FUNCTION_BLOCK FB_ProcessSimulation
VAR_INPUT
	bEnable: BOOL;
	
	bRotateTable: BOOL;
	bLinearSliderMoveToPick : BOOL;
	bLinearSliderMoveToPlace : BOOL;
	
	tPartSensorDelay: TIME;
	tLinearSliderPickPosSensorDelay : TIME;
	tLinearSliderPlacePosSensorDelay : TIME;
END_VAR
VAR_OUTPUT
	bPartSensorSignal: BOOL;
	bLinearSliderPickPosSensorSignal: BOOL;
	bLinearSliderPlacePosSensorSignal: BOOL; 
END_VAR
VAR
	fbPartSensorDelayTmr: TON;
	fbLinearSliderPickPosSensorDelayTmr: TON;
	fbLinearSliderPlacePosSensorDelayTmr: TON;
END_VAR

fbPartSensorDelayTmr(IN:= bEnable AND bRotateTable, 
					PT:= tPartSensorDelay, 
					Q=> bPartSensorSignal, ET=> );
					
fbLinearSliderPickPosSensorDelayTmr(IN:= bEnable AND bLinearSliderMoveToPick, 
									PT:= tLinearSliderPickPosSensorDelay, 
									Q=> bLinearSliderPickPosSensorSignal, ET=> );
									
fbLinearSliderPlacePosSensorDelayTmr(IN:= bEnable AND bLinearSliderMoveToPlace, 
									PT:= tLinearSliderPlacePosSensorDelay, 
									Q=> bLinearSliderPlacePosSensorSignal, ET=> );

END_FUNCTION_BLOCK

(* stored: Version 1.1.0.1, ProductVersion 3.1.4024.12
   POU FB_ProcessSimulation: Id {d0951dc2-7fe7-4eb0-9a9c-218b7ed9d559}, SpecialFunc None *)
